// TIA Portal V16 export
// export: Created 2021-07-12T14:47:14.0696887Z, ExportSetting WithDefaults, DisplayName Totally Integrated Automation Portal, DisplayVersion V16, DisplayName TIA Portal Version Control Interface, DisplayVersion V16, DisplayName TIA Portal Openness, DisplayVersion V16, DisplayName STEP 7 Professional, DisplayVersion V16, DisplayName STEP 7 Safety, DisplayVersion V16, DisplayName WinCC Professional, DisplayVersion V16
ORGANIZATION_BLOCK "MC-PostServo"   // OB95, LAD, PostServo
{ S7_Optimized_Access := 'TRUE' }
VERSION : 0.1
// stored: IsIECCheckEnabled false, SetENOAutomatically false
   VAR_INPUT
      Initial_Call : Bool;
      PIP_Input : Bool;
      PIP_Output : Bool;
      IO_System : USInt;
      Event_Count : Int;
      Synchronous : Bool;
      CycleTime : UDInt;
   END_VAR
   VAR_TEMP
      tempCycleTime : LReal;
      tempCycleTimeLINT : LInt;
      tempRetVal : Word;
      VELOO : Real;
      cetvel2 : Real;
   END_VAR
   VAR_TEMP   // added for the SCL form of the ladder/FBD networks
      _w1 : Bool;
      _w2 : Bool;
   END_VAR
BEGIN

REGION Network 1: Set characteristics of axis at first call
   // Initial setting of valve characteristics.
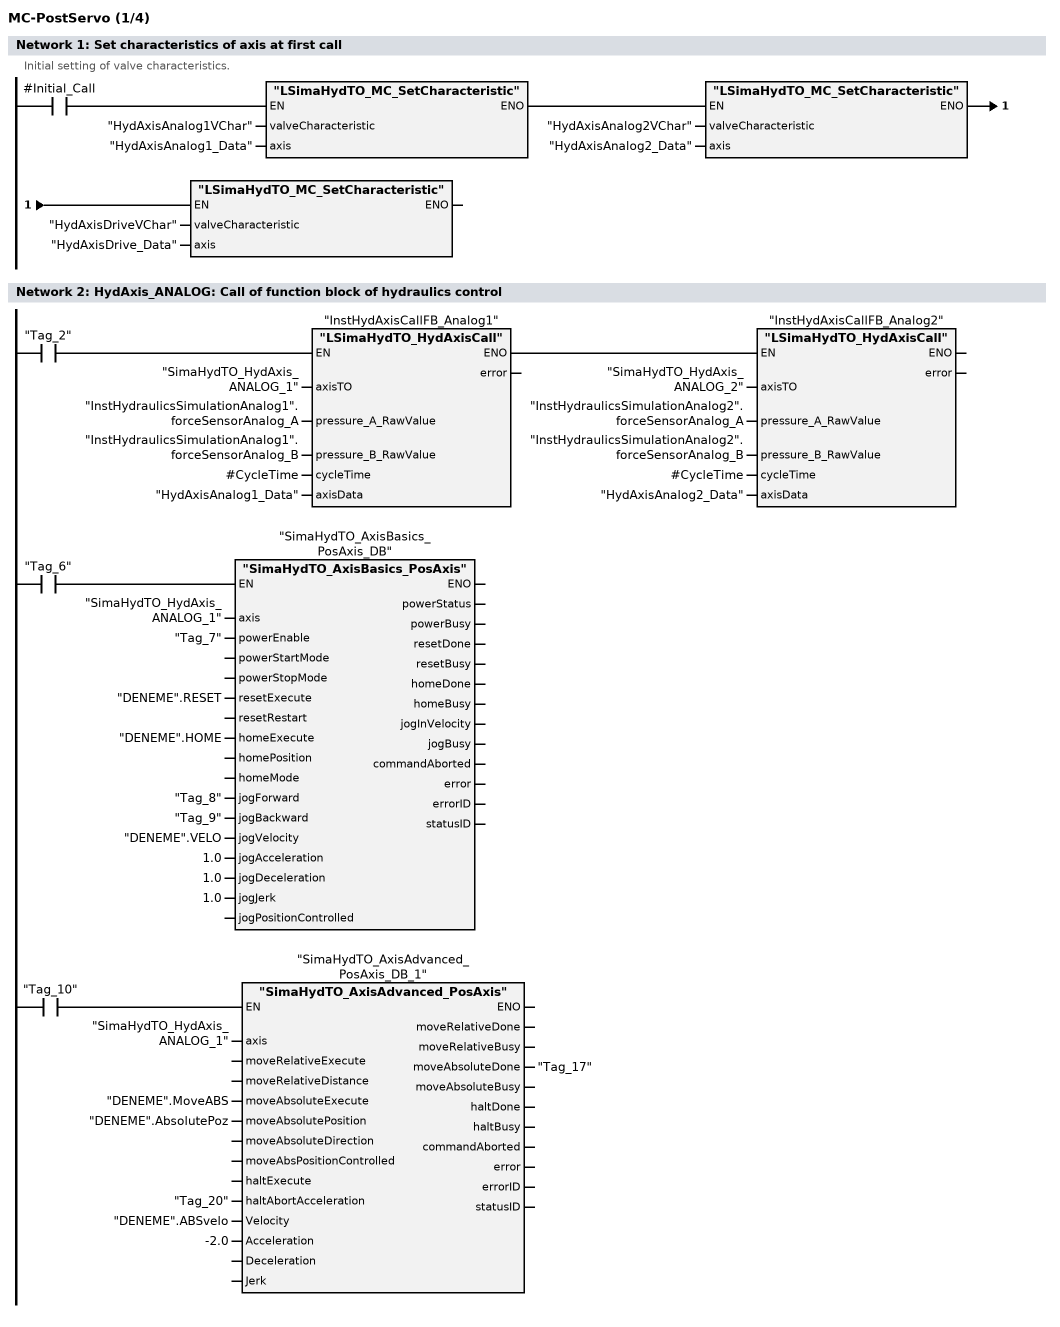
   RUNG wire#powerrail
      Contact( #Initial_Call )
      "LSimaHydTO_MC_SetCharacteristic"(valveCharacteristic := "HydAxisAnalog1VChar", axis := "HydAxisAnalog1_Data")
      "LSimaHydTO_MC_SetCharacteristic"(valveCharacteristic := "HydAxisAnalog2VChar", axis := "HydAxisAnalog2_Data")
      "LSimaHydTO_MC_SetCharacteristic"(valveCharacteristic := "HydAxisDriveVChar", axis := "HydAxisDrive_Data")
   END_RUNG
   // the same network as SCL:
   "LSimaHydTO_MC_SetCharacteristic"(EN := #Initial_Call,
                           valveCharacteristic := "HydAxisAnalog1VChar",
                           axis := "HydAxisAnalog1_Data",
                           ENO => #_w1);
   "LSimaHydTO_MC_SetCharacteristic"(EN := #_w1,
                           valveCharacteristic := "HydAxisAnalog2VChar",
                           axis := "HydAxisAnalog2_Data",
                           ENO => #_w2);
   IF #_w2 THEN
       "LSimaHydTO_MC_SetCharacteristic"(valveCharacteristic := "HydAxisDriveVChar", axis := "HydAxisDrive_Data");
   END_IF;
END_REGION

REGION Network 2: HydAxis_ANALOG: Call of function block of hydraulics control
   RUNG wire#powerrail
      Contact( "Tag_2" )
      "InstHydAxisCallFB_Analog1"(axisTO := "SimaHydTO_HydAxis_ANALOG_1", pressure_A_RawValue := "InstHydraulicsSimulationAnalog1".forceSensorAnalog_A, pressure_B_RawValue := "InstHydraulicsSimulationAnalog1".forceSensorAnalog_B, cycleTime := #CycleTime, axisData := "HydAxisAnalog1_Data", error =>)
      "InstHydAxisCallFB_Analog2"(axisTO := "SimaHydTO_HydAxis_ANALOG_2", pressure_A_RawValue := "InstHydraulicsSimulationAnalog2".forceSensorAnalog_A, pressure_B_RawValue := "InstHydraulicsSimulationAnalog2".forceSensorAnalog_B, cycleTime := #CycleTime, axisData := "HydAxisAnalog2_Data", error =>)
   END_RUNG
   RUNG wire#powerrail
      Contact( "Tag_6" )
      "SimaHydTO_AxisBasics_PosAxis_DB"(axis := "SimaHydTO_HydAxis_ANALOG_1", powerEnable := "Tag_7", powerStartMode :=, powerStopMode :=, resetExecute := "DENEME".RESET, resetRestart :=, homeExecute := "DENEME".HOME, homePosition :=, homeMode :=, jogForward := "Tag_8", jogBackward := "Tag_9", jogVelocity := "DENEME".VELO, jogAcceleration := 1.0, jogDeceleration := 1.0, jogJerk := 1.0, jogPositionControlled :=, powerStatus =>, powerBusy =>, resetDone =>, resetBusy =>, homeDone =>, homeBusy =>, jogInVelocity =>, jogBusy =>, commandAborted =>, error =>, errorID =>, statusID =>)
   END_RUNG
   RUNG wire#powerrail
      Contact( "Tag_10" )
      "SimaHydTO_AxisAdvanced_PosAxis_DB_1"(axis := "SimaHydTO_HydAxis_ANALOG_1", moveRelativeExecute :=, moveRelativeDistance :=, moveAbsoluteExecute := "DENEME".MoveABS, moveAbsolutePosition := "DENEME".AbsolutePoz, moveAbsoluteDirection :=, moveAbsPositionControlled :=, haltExecute :=, haltAbortAcceleration := "Tag_20", Velocity := "DENEME".ABSvelo, Acceleration := -2.0, Deceleration :=, Jerk :=, moveRelativeDone =>, moveRelativeBusy =>, moveAbsoluteDone => "Tag_17", moveAbsoluteBusy =>, haltDone =>, haltBusy =>, commandAborted =>, error =>, errorID =>, statusID =>)
   END_RUNG
   // the same network as SCL:
   "InstHydAxisCallFB_Analog1"(EN := "Tag_2",   // "LSimaHydTO_HydAxisCall"
                           axisTO := "SimaHydTO_HydAxis_ANALOG_1",
                           pressure_A_RawValue := "InstHydraulicsSimulationAnalog1".forceSensorAnalog_A,
                           pressure_B_RawValue := "InstHydraulicsSimulationAnalog1".forceSensorAnalog_B,
                           cycleTime := #CycleTime,
                           axisData := "HydAxisAnalog1_Data",
                           ENO => #_w1);
   IF #_w1 THEN
       "InstHydAxisCallFB_Analog2"(axisTO := "SimaHydTO_HydAxis_ANALOG_2",   // "LSimaHydTO_HydAxisCall"
                               pressure_A_RawValue := "InstHydraulicsSimulationAnalog2".forceSensorAnalog_A,
                               pressure_B_RawValue := "InstHydraulicsSimulationAnalog2".forceSensorAnalog_B,
                               cycleTime := #CycleTime,
                               axisData := "HydAxisAnalog2_Data");
   END_IF;
   IF "Tag_6" THEN
       "SimaHydTO_AxisBasics_PosAxis_DB"(axis := "SimaHydTO_HydAxis_ANALOG_1",   // "SimaHydTO_AxisBasics_PosAxis"
                               powerEnable := "Tag_7",
                               resetExecute := "DENEME".RESET,
                               homeExecute := "DENEME".HOME,
                               jogForward := "Tag_8",
                               jogBackward := "Tag_9",
                               jogVelocity := "DENEME".VELO,
                               jogAcceleration := 1.0,
                               jogDeceleration := 1.0,
                               jogJerk := 1.0);
   END_IF;
   IF "Tag_10" THEN
       "SimaHydTO_AxisAdvanced_PosAxis_DB_1"(axis := "SimaHydTO_HydAxis_ANALOG_1",   // "SimaHydTO_AxisAdvanced_PosAxis"
                               moveAbsoluteExecute := "DENEME".MoveABS,
                               moveAbsolutePosition := "DENEME".AbsolutePoz,
                               haltAbortAcceleration := "Tag_20",
                               Velocity := "DENEME".ABSvelo,
                               Acceleration := -2.0,
                               moveAbsoluteDone => "Tag_17");
   END_IF;
END_REGION

REGION Network 3: HydAxis_ANALOG: Call of function block of hydraulics axis simulation
   // The simulation uses as input signal "analogInput" the real output integer value of analog module AQ. (-27648...+27648)
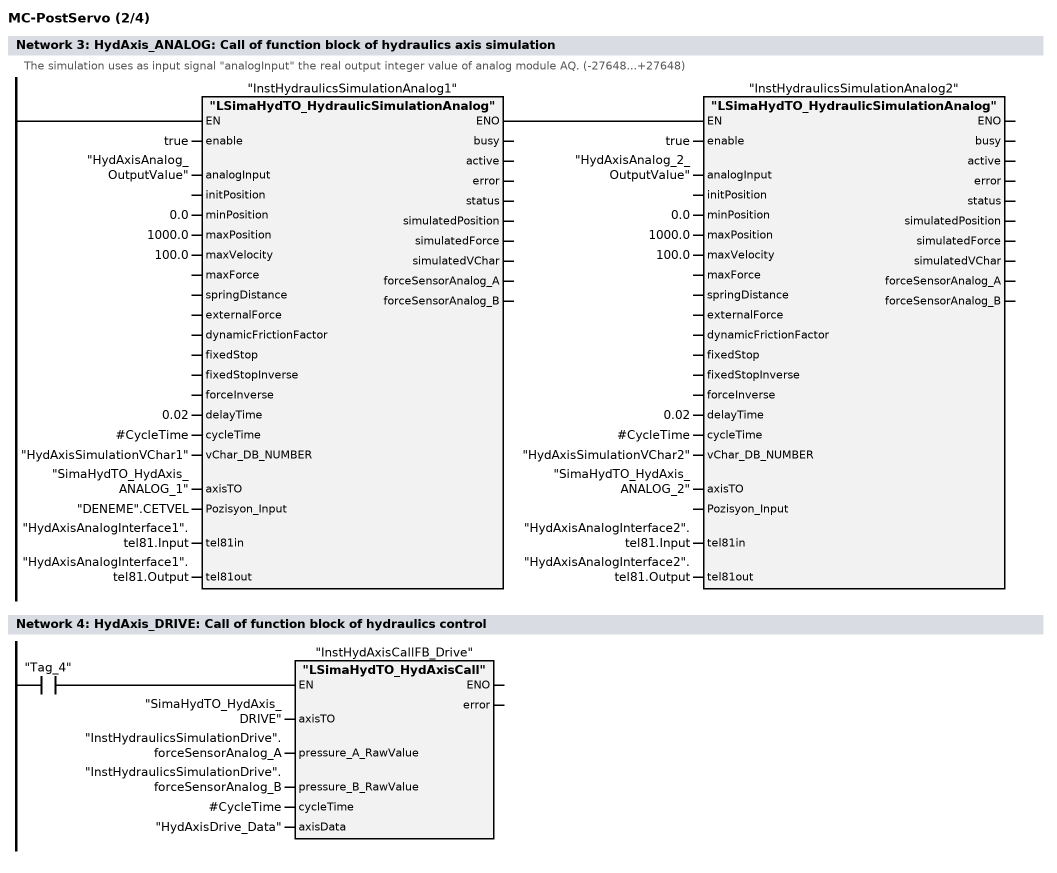
   RUNG wire#powerrail
      "InstHydraulicsSimulationAnalog1"(enable := true, analogInput := "HydAxisAnalog_OutputValue", initPosition :=, minPosition := 0.0, maxPosition := 1000.0, maxVelocity := 100.0, maxForce :=, springDistance :=, externalForce :=, dynamicFrictionFactor :=, fixedStop :=, fixedStopInverse :=, forceInverse :=, delayTime := 0.02, cycleTime := #CycleTime, vChar_DB_NUMBER := "HydAxisSimulationVChar1", axisTO := "SimaHydTO_HydAxis_ANALOG_1", Pozisyon_Input := "DENEME".CETVEL, tel81in := "HydAxisAnalogInterface1".tel81.Input, tel81out := "HydAxisAnalogInterface1".tel81.Output, busy =>, active =>, error =>, status =>, simulatedPosition =>, simulatedForce =>, simulatedVChar =>, forceSensorAnalog_A =>, forceSensorAnalog_B =>)
      "InstHydraulicsSimulationAnalog2"(enable := true, analogInput := "HydAxisAnalog_2_OutputValue", initPosition :=, minPosition := 0.0, maxPosition := 1000.0, maxVelocity := 100.0, maxForce :=, springDistance :=, externalForce :=, dynamicFrictionFactor :=, fixedStop :=, fixedStopInverse :=, forceInverse :=, delayTime := 0.02, cycleTime := #CycleTime, vChar_DB_NUMBER := "HydAxisSimulationVChar2", axisTO := "SimaHydTO_HydAxis_ANALOG_2", Pozisyon_Input :=, tel81in := "HydAxisAnalogInterface2".tel81.Input, tel81out := "HydAxisAnalogInterface2".tel81.Output, busy =>, active =>, error =>, status =>, simulatedPosition =>, simulatedForce =>, simulatedVChar =>, forceSensorAnalog_A =>, forceSensorAnalog_B =>)
   END_RUNG
   // the same network as SCL:
   "InstHydraulicsSimulationAnalog1"(enable := true,   // "LSimaHydTO_HydraulicSimulationAnalog"
                           analogInput := "HydAxisAnalog_OutputValue",
                           minPosition := 0.0,
                           maxPosition := 1000.0,
                           maxVelocity := 100.0,
                           delayTime := 0.02,
                           cycleTime := #CycleTime,
                           vChar_DB_NUMBER := "HydAxisSimulationVChar1",
                           axisTO := "SimaHydTO_HydAxis_ANALOG_1",
                           Pozisyon_Input := "DENEME".CETVEL,
                           tel81in := "HydAxisAnalogInterface1".tel81.Input,
                           tel81out := "HydAxisAnalogInterface1".tel81.Output,
                           ENO => #_w1);
   IF #_w1 THEN
       "InstHydraulicsSimulationAnalog2"(enable := true,   // "LSimaHydTO_HydraulicSimulationAnalog"
                               analogInput := "HydAxisAnalog_2_OutputValue",
                               minPosition := 0.0,
                               maxPosition := 1000.0,
                               maxVelocity := 100.0,
                               delayTime := 0.02,
                               cycleTime := #CycleTime,
                               vChar_DB_NUMBER := "HydAxisSimulationVChar2",
                               axisTO := "SimaHydTO_HydAxis_ANALOG_2",
                               tel81in := "HydAxisAnalogInterface2".tel81.Input,
                               tel81out := "HydAxisAnalogInterface2".tel81.Output);
   END_IF;
END_REGION

REGION Network 4: HydAxis_DRIVE: Call of function block of hydraulics control
   RUNG wire#powerrail
      Contact( "Tag_4" )
      "InstHydAxisCallFB_Drive"(axisTO := "SimaHydTO_HydAxis_DRIVE", pressure_A_RawValue := "InstHydraulicsSimulationDrive".forceSensorAnalog_A, pressure_B_RawValue := "InstHydraulicsSimulationDrive".forceSensorAnalog_B, cycleTime := #CycleTime, axisData := "HydAxisDrive_Data", error =>)
   END_RUNG
   // the same network as SCL:
   IF "Tag_4" THEN
       "InstHydAxisCallFB_Drive"(axisTO := "SimaHydTO_HydAxis_DRIVE",   // "LSimaHydTO_HydAxisCall"
                               pressure_A_RawValue := "InstHydraulicsSimulationDrive".forceSensorAnalog_A,
                               pressure_B_RawValue := "InstHydraulicsSimulationDrive".forceSensorAnalog_B,
                               cycleTime := #CycleTime,
                               axisData := "HydAxisDrive_Data");
   END_IF;
END_REGION

REGION Network 5: HydAxis_DRIVE: Call of function block of hydraulics axis simulation
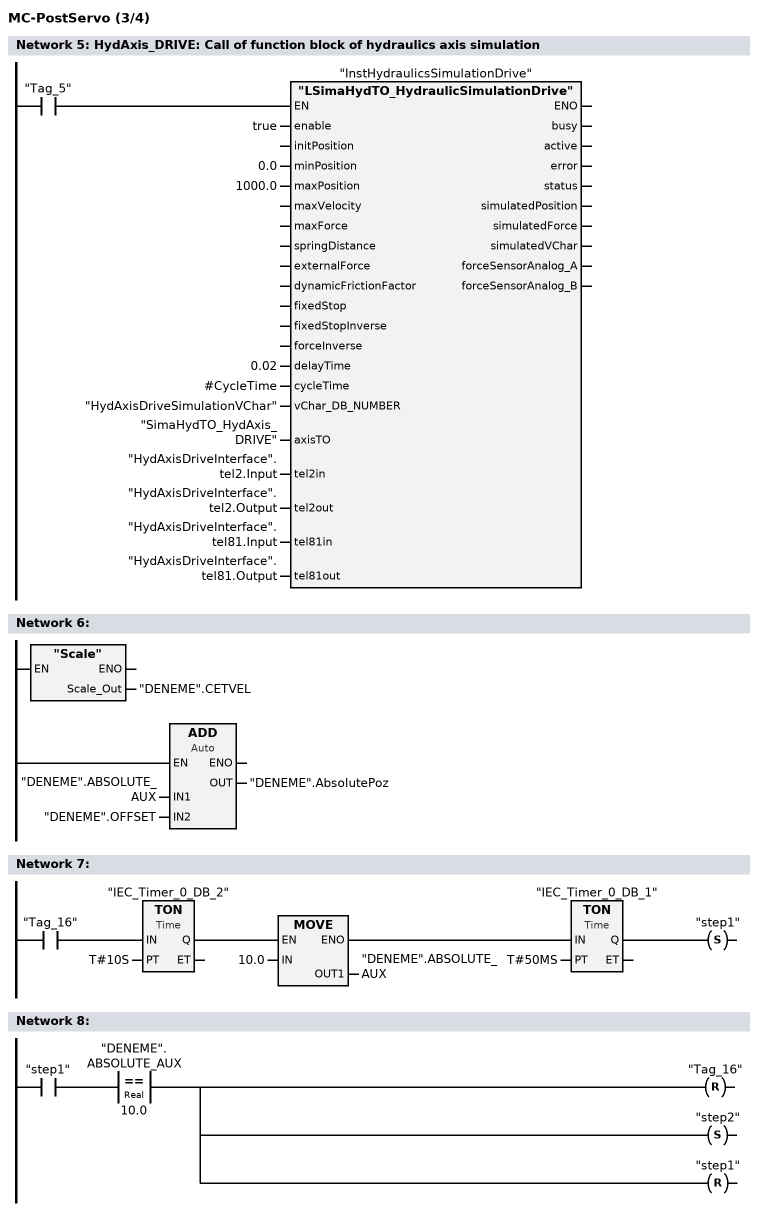
   RUNG wire#powerrail
      Contact( "Tag_5" )
      "InstHydraulicsSimulationDrive"(enable := true, initPosition :=, minPosition := 0.0, maxPosition := 1000.0, maxVelocity :=, maxForce :=, springDistance :=, externalForce :=, dynamicFrictionFactor :=, fixedStop :=, fixedStopInverse :=, forceInverse :=, delayTime := 0.02, cycleTime := #CycleTime, vChar_DB_NUMBER := "HydAxisDriveSimulationVChar", axisTO := "SimaHydTO_HydAxis_DRIVE", tel2in := "HydAxisDriveInterface".tel2.Input, tel2out := "HydAxisDriveInterface".tel2.Output, tel81in := "HydAxisDriveInterface".tel81.Input, tel81out := "HydAxisDriveInterface".tel81.Output, busy =>, active =>, error =>, status =>, simulatedPosition =>, simulatedForce =>, simulatedVChar =>, forceSensorAnalog_A =>, forceSensorAnalog_B =>)
   END_RUNG
   // the same network as SCL:
   IF "Tag_5" THEN
       "InstHydraulicsSimulationDrive"(enable := true,   // "LSimaHydTO_HydraulicSimulationDrive"
                               minPosition := 0.0,
                               maxPosition := 1000.0,
                               delayTime := 0.02,
                               cycleTime := #CycleTime,
                               vChar_DB_NUMBER := "HydAxisDriveSimulationVChar",
                               axisTO := "SimaHydTO_HydAxis_DRIVE",
                               tel2in := "HydAxisDriveInterface".tel2.Input,
                               tel2out := "HydAxisDriveInterface".tel2.Output,
                               tel81in := "HydAxisDriveInterface".tel81.Input,
                               tel81out := "HydAxisDriveInterface".tel81.Output);
   END_IF;
END_REGION

REGION Network 6
   RUNG wire#powerrail
      "Scale"(Scale_Out => "DENEME".CETVEL)
   END_RUNG
   RUNG wire#powerrail
      Add(in1 := "DENEME".ABSOLUTE_AUX, in2 := "DENEME".OFFSET, out => "DENEME".AbsolutePoz)
   END_RUNG
   // the same network as SCL:
   "Scale"(Scale_Out => "DENEME".CETVEL);
   "DENEME".AbsolutePoz := "DENEME".ABSOLUTE_AUX + "DENEME".OFFSET;
END_REGION

REGION Network 7
   RUNG wire#powerrail
      Contact( "Tag_16" )
      { S7_Templates := "time_type := Time" } "IEC_Timer_0_DB_2".TON(pt := T#10S, et =>)
      Move(in := 10.0, out1 => "DENEME".ABSOLUTE_AUX)
      { S7_Templates := "time_type := Time" } "IEC_Timer_0_DB_1".TON(pt := T#50MS, et =>)
      S_Coil( "step1" )
   END_RUNG
   // the same network as SCL:
   "IEC_Timer_0_DB_2".TON(IN := "Tag_16", PT := T#10S);
   IF "IEC_Timer_0_DB_2".Q THEN "DENEME".ABSOLUTE_AUX := 10.0; END_IF;
   "IEC_Timer_0_DB_1".TON(IN := "IEC_Timer_0_DB_2".Q, PT := T#50MS);
   IF "IEC_Timer_0_DB_1".Q THEN "step1" := TRUE; END_IF;
END_REGION

REGION Network 8
   RUNG wire#powerrail
      Contact( "step1" )
      { S7_Templates := "SrcType := Real" } EQ_Contact(in1 := "DENEME".ABSOLUTE_AUX, in2 := 10.0)
      wire#w1
      R_Coil( "Tag_16" )
   END_RUNG
   RUNG wire#w1
      S_Coil( "step2" )
   END_RUNG
   RUNG wire#w1
      R_Coil( "step1" )
   END_RUNG
   // the same network as SCL:
   IF "step1" AND ("DENEME".ABSOLUTE_AUX = 10.0) THEN
       "Tag_16" := FALSE;
       "step2" := TRUE;
       "step1" := FALSE;
   END_IF;
END_REGION

REGION Network 9
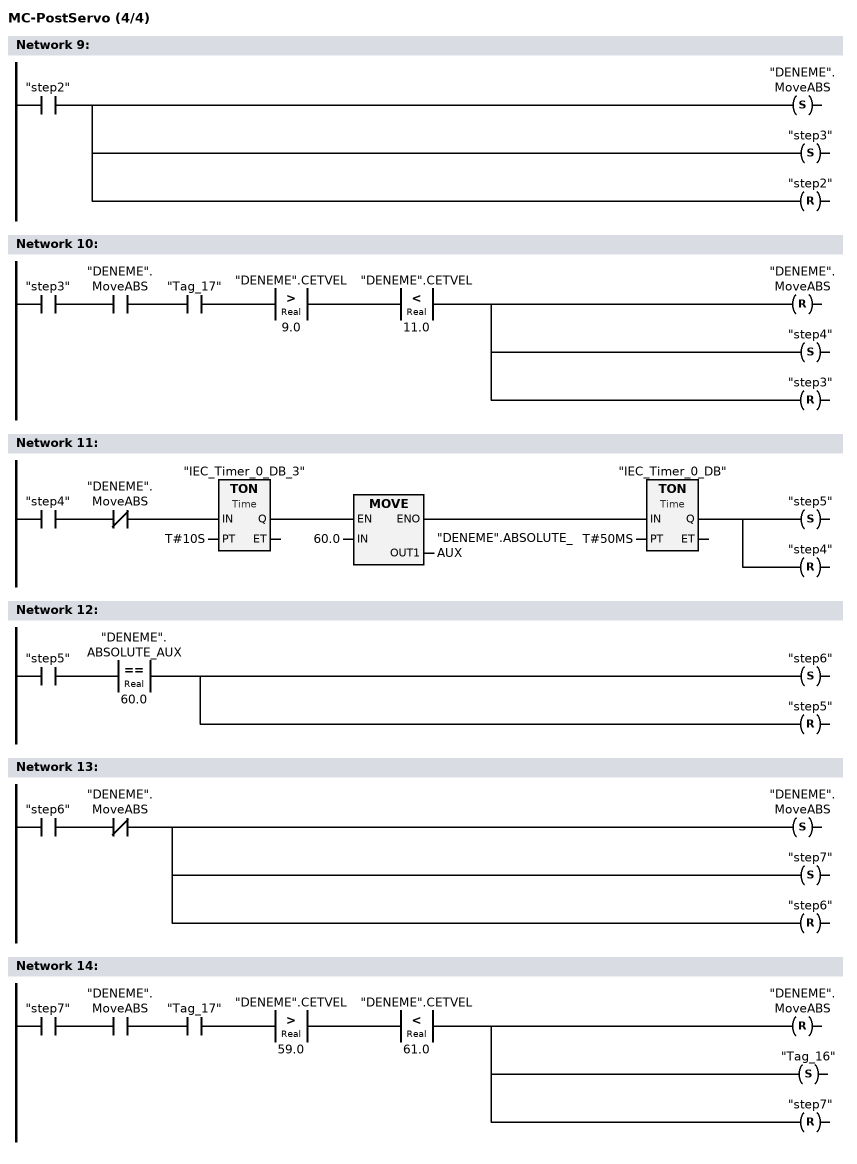
   RUNG wire#powerrail
      Contact( "step2" )
      wire#w1
      S_Coil( "DENEME".MoveABS )
   END_RUNG
   RUNG wire#w1
      S_Coil( "step3" )
   END_RUNG
   RUNG wire#w1
      R_Coil( "step2" )
   END_RUNG
   // the same network as SCL:
   IF "step2" THEN
       "DENEME".MoveABS := TRUE;
       "step3" := TRUE;
       "step2" := FALSE;
   END_IF;
END_REGION

REGION Network 10
   RUNG wire#powerrail
      Contact( "step3" )
      Contact( "DENEME".MoveABS )
      Contact( "Tag_17" )
      { S7_Templates := "SrcType := Real" } GT_Contact(in1 := "DENEME".CETVEL, in2 := 9.0)
      { S7_Templates := "SrcType := Real" } LT_Contact(in1 := "DENEME".CETVEL, in2 := 11.0)
      wire#w1
      R_Coil( "DENEME".MoveABS )
   END_RUNG
   RUNG wire#w1
      S_Coil( "step4" )
   END_RUNG
   RUNG wire#w1
      R_Coil( "step3" )
   END_RUNG
   // the same network as SCL:
   #_w1 := "step3" AND "DENEME".MoveABS AND "Tag_17" AND ("DENEME".CETVEL > 9.0) AND ("DENEME".CETVEL < 11.0);
   IF #_w1 THEN
       "DENEME".MoveABS := FALSE;
       "step4" := TRUE;
       "step3" := FALSE;
   END_IF;
END_REGION

REGION Network 11
   RUNG wire#powerrail
      Contact( "step4" )
      I_Contact( "DENEME".MoveABS )
      { S7_Templates := "time_type := Time" } "IEC_Timer_0_DB_3".TON(pt := T#10S, et =>)
      Move(in := 60.0, out1 => "DENEME".ABSOLUTE_AUX)
      { S7_Templates := "time_type := Time" } "IEC_Timer_0_DB".TON(pt := T#50MS, et =>)
      wire#w1
      S_Coil( "step5" )
   END_RUNG
   RUNG wire#w1
      R_Coil( "step4" )
   END_RUNG
   // the same network as SCL:
   "IEC_Timer_0_DB_3".TON(IN := "step4" AND NOT "DENEME".MoveABS, PT := T#10S);
   IF "IEC_Timer_0_DB_3".Q THEN "DENEME".ABSOLUTE_AUX := 60.0; END_IF;
   "IEC_Timer_0_DB".TON(IN := "IEC_Timer_0_DB_3".Q, PT := T#50MS);
   IF "IEC_Timer_0_DB".Q THEN
       "step5" := TRUE;
       "step4" := FALSE;
   END_IF;
END_REGION

REGION Network 12
   RUNG wire#powerrail
      Contact( "step5" )
      { S7_Templates := "SrcType := Real" } EQ_Contact(in1 := "DENEME".ABSOLUTE_AUX, in2 := 60.0)
      wire#w1
      S_Coil( "step6" )
   END_RUNG
   RUNG wire#w1
      R_Coil( "step5" )
   END_RUNG
   // the same network as SCL:
   IF "step5" AND ("DENEME".ABSOLUTE_AUX = 60.0) THEN
       "step6" := TRUE;
       "step5" := FALSE;
   END_IF;
END_REGION

REGION Network 13
   RUNG wire#powerrail
      Contact( "step6" )
      I_Contact( "DENEME".MoveABS )
      wire#w1
      S_Coil( "DENEME".MoveABS )
   END_RUNG
   RUNG wire#w1
      S_Coil( "step7" )
   END_RUNG
   RUNG wire#w1
      R_Coil( "step6" )
   END_RUNG
   // the same network as SCL:
   #_w1 := "step6" AND NOT "DENEME".MoveABS;
   IF #_w1 THEN
       "DENEME".MoveABS := TRUE;
       "step7" := TRUE;
       "step6" := FALSE;
   END_IF;
END_REGION

REGION Network 14
   RUNG wire#powerrail
      Contact( "step7" )
      Contact( "DENEME".MoveABS )
      Contact( "Tag_17" )
      { S7_Templates := "SrcType := Real" } GT_Contact(in1 := "DENEME".CETVEL, in2 := 59.0)
      { S7_Templates := "SrcType := Real" } LT_Contact(in1 := "DENEME".CETVEL, in2 := 61.0)
      wire#w1
      R_Coil( "DENEME".MoveABS )
   END_RUNG
   RUNG wire#w1
      S_Coil( "Tag_16" )
   END_RUNG
   RUNG wire#w1
      R_Coil( "step7" )
   END_RUNG
   // the same network as SCL:
   #_w1 := "step7" AND "DENEME".MoveABS AND "Tag_17" AND ("DENEME".CETVEL > 59.0) AND ("DENEME".CETVEL < 61.0);
   IF #_w1 THEN
       "DENEME".MoveABS := FALSE;
       "Tag_16" := TRUE;
       "step7" := FALSE;
   END_IF;
END_REGION
END_ORGANIZATION_BLOCK
